PROGRAM C04_ContolButtons

VAR
	rtrigStartButton		:   	R_TRIG;
    	ftrigStartButton		:   	F_TRIG;
    	rtrigResetButton		:   	R_TRIG;
    	ftrigResetButton		:   	F_TRIG;
    	rtrigStopButton		:   	R_TRIG;
	ftrigStopButton			:   	F_TRIG;
	tpShortResetPulse		:	TP;
	tofLongResetPulse		:	TOF;
	tonForceResetSignal		:	TON;

	fbHardResetTimer		:	FB_LongShortPress;

	aLabelPrintButton		: ARRAY[1..cMAX_PRINTER_NUMBER] OF  R_TRIG;
	aLabelApplyButton		: ARRAY[1..cMAX_PRINTER_NUMBER] OF  R_TRIG;

	rtrigResetTCPServer		:   	R_TRIG;
    	ftrigResetTCPServer		:   	F_TRIG;

END_VAR

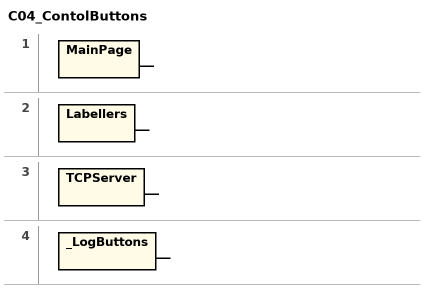
// NETWORK 1
MainPage();

// NETWORK 2
Labellers();

// NETWORK 3
TCPServer();

// NETWORK 4
_LogButtons();

ACTION _LogButtons:
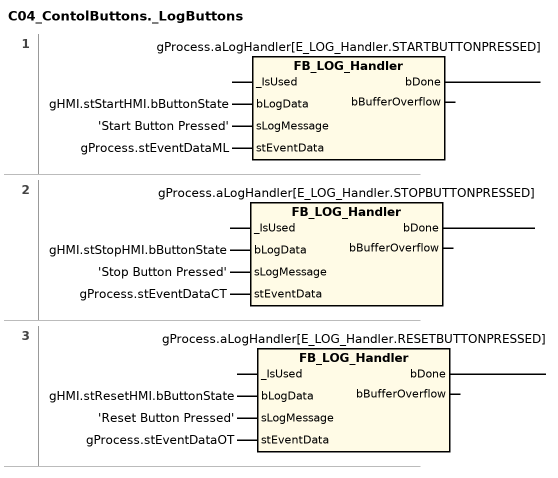
// NETWORK 1
gProcess.aLogHandler[E_LOG_Handler.STARTBUTTONPRESSED](
    bLogData := gHMI.stStartHMI.bButtonState,
    sLogMessage := 'Start Button Pressed',
    stEventData := gProcess.stEventDataML); // FB_LOG_Handler

// NETWORK 2
gProcess.aLogHandler[E_LOG_Handler.STOPBUTTONPRESSED](
    bLogData := gHMI.stStopHMI.bButtonState,
    sLogMessage := 'Stop Button Pressed',
    stEventData := gProcess.stEventDataCT); // FB_LOG_Handler

// NETWORK 3
gProcess.aLogHandler[E_LOG_Handler.RESETBUTTONPRESSED](
    bLogData := gHMI.stResetHMI.bButtonState,
    sLogMessage := 'Reset Button Pressed',
    stEventData := gProcess.stEventDataOT); // FB_LOG_Handler
END_ACTION

ACTION Labellers:
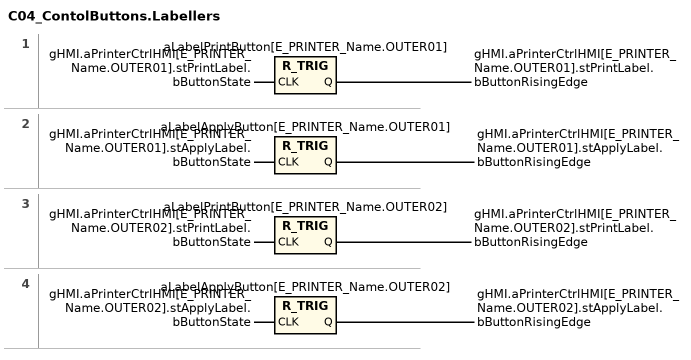
// NETWORK 1
aLabelPrintButton[E_PRINTER_Name.OUTER01](CLK := gHMI.aPrinterCtrlHMI[E_PRINTER_Name.OUTER01].stPrintLabel.bButtonState); // R_TRIG
gHMI.aPrinterCtrlHMI[E_PRINTER_Name.OUTER01].stPrintLabel.bButtonRisingEdge := aLabelPrintButton[E_PRINTER_Name.OUTER01].Q;

// NETWORK 2
aLabelApplyButton[E_PRINTER_Name.OUTER01](CLK := gHMI.aPrinterCtrlHMI[E_PRINTER_Name.OUTER01].stApplyLabel.bButtonState); // R_TRIG
gHMI.aPrinterCtrlHMI[E_PRINTER_Name.OUTER01].stApplyLabel.bButtonRisingEdge := aLabelApplyButton[E_PRINTER_Name.OUTER01].Q;

// NETWORK 3
aLabelPrintButton[E_PRINTER_Name.OUTER02](CLK := gHMI.aPrinterCtrlHMI[E_PRINTER_Name.OUTER02].stPrintLabel.bButtonState); // R_TRIG
gHMI.aPrinterCtrlHMI[E_PRINTER_Name.OUTER02].stPrintLabel.bButtonRisingEdge := aLabelPrintButton[E_PRINTER_Name.OUTER02].Q;

// NETWORK 4
aLabelApplyButton[E_PRINTER_Name.OUTER02](CLK := gHMI.aPrinterCtrlHMI[E_PRINTER_Name.OUTER02].stApplyLabel.bButtonState); // R_TRIG
gHMI.aPrinterCtrlHMI[E_PRINTER_Name.OUTER02].stApplyLabel.bButtonRisingEdge := aLabelApplyButton[E_PRINTER_Name.OUTER02].Q;
END_ACTION

ACTION MainPage:
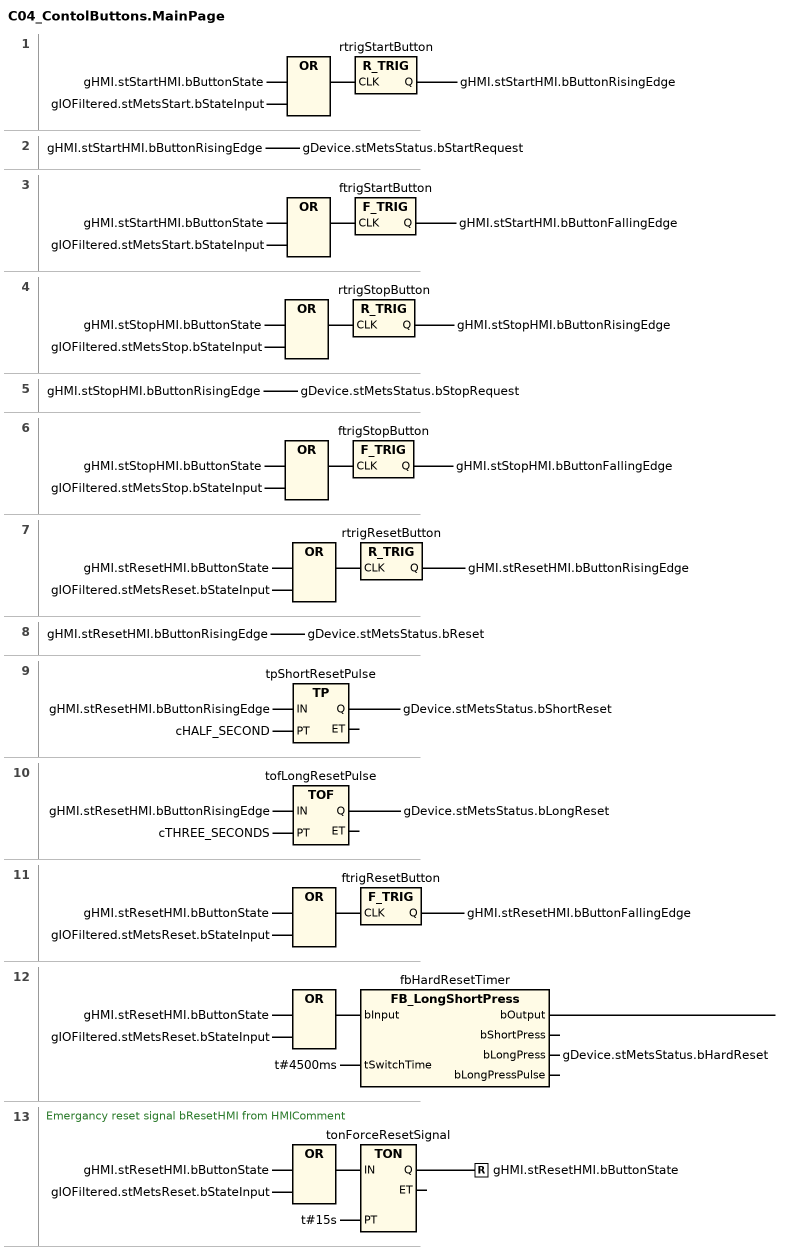
// NETWORK 1
rtrigStartButton(CLK := gHMI.stStartHMI.bButtonState OR gIOFiltered.stMetsStart.bStateInput); // R_TRIG
gHMI.stStartHMI.bButtonRisingEdge := rtrigStartButton.Q;

// NETWORK 2
gDevice.stMetsStatus.bStartRequest := gHMI.stStartHMI.bButtonRisingEdge;

// NETWORK 3
ftrigStartButton(CLK := gHMI.stStartHMI.bButtonState OR gIOFiltered.stMetsStart.bStateInput); // F_TRIG
gHMI.stStartHMI.bButtonFallingEdge := ftrigStartButton.Q;

// NETWORK 4
rtrigStopButton(CLK := gHMI.stStopHMI.bButtonState OR gIOFiltered.stMetsStop.bStateInput); // R_TRIG
gHMI.stStopHMI.bButtonRisingEdge := rtrigStopButton.Q;

// NETWORK 5
gDevice.stMetsStatus.bStopRequest := gHMI.stStopHMI.bButtonRisingEdge;

// NETWORK 6
ftrigStopButton(CLK := gHMI.stStopHMI.bButtonState OR gIOFiltered.stMetsStop.bStateInput); // F_TRIG
gHMI.stStopHMI.bButtonFallingEdge := ftrigStopButton.Q;

// NETWORK 7
rtrigResetButton(CLK := gHMI.stResetHMI.bButtonState OR gIOFiltered.stMetsReset.bStateInput); // R_TRIG
gHMI.stResetHMI.bButtonRisingEdge := rtrigResetButton.Q;

// NETWORK 8
gDevice.stMetsStatus.bReset := gHMI.stResetHMI.bButtonRisingEdge;

// NETWORK 9
tpShortResetPulse(IN := gHMI.stResetHMI.bButtonRisingEdge, PT := cHALF_SECOND); // TP
gDevice.stMetsStatus.bShortReset := tpShortResetPulse.Q;

// NETWORK 10
tofLongResetPulse(IN := gHMI.stResetHMI.bButtonRisingEdge, PT := cTHREE_SECONDS); // TOF
gDevice.stMetsStatus.bLongReset := tofLongResetPulse.Q;

// NETWORK 11
ftrigResetButton(CLK := gHMI.stResetHMI.bButtonState OR gIOFiltered.stMetsReset.bStateInput); // F_TRIG
gHMI.stResetHMI.bButtonFallingEdge := ftrigResetButton.Q;

// NETWORK 12
fbHardResetTimer(
    bInput := gHMI.stResetHMI.bButtonState OR gIOFiltered.stMetsReset.bStateInput,
    tSwitchTime := t#4500ms,
    bLongPress => gDevice.stMetsStatus.bHardReset); // FB_LongShortPress

// NETWORK 13
// Emergancy reset signal bResetHMI from HMIComment
tonForceResetSignal(IN := gHMI.stResetHMI.bButtonState OR gIOFiltered.stMetsReset.bStateInput, PT := t#15s); // TON
gHMI.stResetHMI.bButtonState R= tonForceResetSignal.Q;
END_ACTION

ACTION TCPServer:
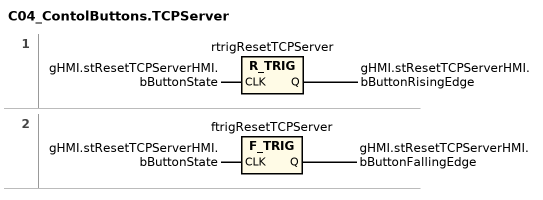
// NETWORK 1
rtrigResetTCPServer(CLK := gHMI.stResetTCPServerHMI.bButtonState); // R_TRIG
gHMI.stResetTCPServerHMI.bButtonRisingEdge := rtrigResetTCPServer.Q;

// NETWORK 2
ftrigResetTCPServer(CLK := gHMI.stResetTCPServerHMI.bButtonState); // F_TRIG
gHMI.stResetTCPServerHMI.bButtonFallingEdge := ftrigResetTCPServer.Q;
END_ACTION

END_PROGRAM

(* stored: Version 1.1.0.1
   POU C04_ContolButtons: Id {556f0493-ceba-4564-96fc-0f2ed8ca213f}, SpecialFunc None
   Action _LogButtons: Id {6ab8737d-2fe5-4726-a2f2-ca627024e493}
   Action Labellers: Id {9320e776-37e6-4a01-8216-254da6246463}
   Action MainPage: Id {69046284-a291-4190-afe4-41499c1e682a}
   Action TCPServer: Id {e4b827f0-4c7e-409f-a7a4-dbd66870841b} *)
